PROGRAM PRG_RecipeManager
VAR
	fbLoadRecipe  	: FB_LoadRecipe;
    fbListFiles  	: FB_ListRecipeFiles;
	fbDeleteRecipe 	: FB_DeleteRecipe;
	fbSaveRecipe 	: FB_SaveRecipe;

    sPrefix      : STRING(64) := 'C:\TwinCAT\Recipes\';
    sFileName    : STRING(255);
	
	bDatagridRowsNaming		 : BOOL := FALSE;
	bClearAvailableFiles	 : BOOL := FALSE;
	bClearAvailableFilesDone : BOOL := FALSE;
	
	
		
	i	: INT;
	
	
END_VAR

VAR_INPUT
	bDatagridToRecipeDone	: BOOL := FALSE;
END_VAR

//Naming the datagrid 1st column with the names in the HMI Recipe Screen just once
IF NOT bDatagridRowsNaming THEN
	ACT_DatagridsRowNaming();
END_IF

// <Load button> ############# Look up for the recipe files in the folder and fill up the GVL_Recipe.aAvailableFiles[]. ######################### 
IF GVL_HMI.bRefreshRecipeList THEN
	//GVL_HMI.bRecipeCorrectLoaded := FALSE;
	//GVL_HMI.bRecipeLoadFailed := FALSE;
	bClearAvailableFiles := TRUE;
	IF bClearAvailableFilesDone THEN
		fbListFiles(bExecute := TRUE);
	END_IF
ELSE
	bClearAvailableFiles := FALSE;
	bClearAvailableFilesDone := FALSE;
    fbListFiles(bExecute := FALSE);
END_IF

// Clear the Available files datagrid in the load file popup
IF bClearAvailableFiles THEN
	ACT_ClearAvailableFiles();
END_IF

// Reset load actions once its done
IF fbListFiles.bDone THEN
	GVL_HMI.bRefreshRecipeList := FALSE;
END_IF

 //Reset file name
sFileName := '';

// Run the loading recipe from selected row in the recipe load popup
sFileName := CONCAT(sPrefix, CONCAT(GVL_Recipe.sSelectedRecipeName, '.json')); // File naming assemble for the selected row in the recipe load popup
fbLoadRecipe( sFileName := sFileName, bExecute := GVL_HMI.bRecipeLoadFromFile AND  DB_Query.timerVD.Q );


IF fbLoadRecipe.bError THEN
	GVL_HMI.bRecipeLoadFailed := TRUE;
	//GVL_HMI.bRecipeLoadFromFile := FALSE;
END_IF

// After the recipe loading, reseting and setting the flags
IF NOT fbLoadRecipe.bBusy AND NOT fbLoadRecipe.bError AND GVL_HMI.bRecipeLoadFromFile AND DB_Query.timerVD.Q THEN
	GVL_HMI.bRecipeCorrectLoaded := TRUE;
	GVL_HMI.bRecipeLoadFromFile := FALSE;
	DB_Query.timerVD(in:= FALSE);
	ACT_ClearStActiveRecipe(); //Clears the Active Recipe
END_IF
// <\Load button> ############# END ##############

// <Save Button> ############# Fill stCurrentRecipe from HMI datagrids if save button is pressed ########################
IF GVL_HMI.bRecipeSaveButton THEN
	ACT_DatagridToRecipe();
	IF bDatagridToRecipeDone THEN
		fbSaveRecipe(bExecute := TRUE, sUser := GVL_HMI.stRecipeInfo.sCreatedBy);
		IF fbSaveRecipe.bDone AND NOT fbSaveRecipe.bError THEN
			GVL_HMI.stRecipeInfo.iRevision := GVL_Recipe.stCurrentRecipe.stInfo.iRevision; //Update the datagrid revision that does not come from the grid
			fbSaveRecipe(bExecute := FALSE);
			GVL_HMI.bRecipeSaveDone := TRUE; //Response Success flag to HMI
			GVL_HMI.bRecipeSaveButton := FALSE;	
			bDatagridToRecipeDone := FALSE;
			ACT_ClearStActiveRecipe(); //Clears the Active Recipe
			ELSE IF fbSaveRecipe.bError THEN
				GVL_HMI.bRecipeSaveError := TRUE; //Response Error flag to HMI
			END_IF
		END_IF
		
	END_IF
END_IF
// <\Save Button> ############# END ########################

// <Cancel Button> ############# Reload the datagrids with the recipe in stCurrentRecipe if the bt cancel is pressed during new recipe ########################
IF GVL_HMI.bReloadRecipeDatagrids THEN
	ACT_RecipeToDatagrid();
END_IF
// <\Cancel Button> ############# END ########################

// <Activate Button> ############# Transfer data from stCurrentRecipe for stActivatedRecipe witch will be used on the cycle  ########################
IF GVL_HMI.bRecipeActivateButton THEN
	GVL_Recipe.stActiveRecipe := GVL_Recipe.stCurrentRecipe; //Only fill stActiveRecipe if button Activate was pressed on hmi. 
	IF GVL_Recipe.stCurrentRecipe.stInfo.sMethodName <> '' THEN
		GVL_HMI.bRecipeActivateDone := TRUE;
		GVL_Recipe.bIsThereRecipeActivated := TRUE;
	ELSE
		GVL_HMI.bRecipeActivateError := TRUE;
	END_IF
	
END_IF
// <\Activate Button> ############# END ########################

// <Delete Button> ############# Moves the loaded Recipe file from the root folder for the _deleted folder ########################
IF GVL_HMI.bDeleteRecipeButton THEN
	ACT_PopulateDeleteRecipeInfo();
	GVL_HMI.bDeleteRecipeDone := FALSE;
	GVL_HMI.bDeleteRecipeError := FALSE;
END_IF

fbDeleteRecipe(bExecute := GVL_HMI.bDeleteRecipeConfirm, stFileInfo := GVL_HMI.stDeleteRecipeInfo);

IF fbDeleteRecipe.bDone THEN
	IF NOT fbDeleteRecipe.bError THEN 
		ACT_ClearStCurrentRecipe();
		ACT_ClearHMIDatagrids();
		ACT_ClearStActiveRecipe(); //Clears the Active Recipe
		GVL_HMI.bDeleteRecipeConfirm := FALSE;
		GVL_HMI.bDeleteRecipeDone := TRUE;
	ELSE 
		GVL_HMI.bDeleteRecipeError := TRUE;
	END_IF
END_IF

// <\Delete Button> ############# END ########################

ACTION ACT_ClearAvailableFiles:
//Clear the GVL_Recipe.aAvailableFiles, witch is the list files datagrid data source
IF NOT bClearAvailableFilesDone THEN
	FOR i := 1 TO 50 DO
		GVL_HMI.aAvailableFiles[i].sFileName := '';
		GVL_HMI.aAvailableFiles[i].sMethodName := '';
		GVL_HMI.aAvailableFiles[i].sCreatedBy := '';
		GVL_HMI.aAvailableFiles[i].iRevision := 0;
		GVL_HMI.aAvailableFiles[i].dtLastModified := DT#1970-01-01-00:00;
		GVL_HMI.aAvailableFiles[i].dCreationDate := D#1970-01-01;
	END_FOR
	
	IF i >= 50 THEN
		bClearAvailableFilesDone := TRUE;
	END_IF
END_IF
END_ACTION

ACTION ACT_ClearHMIDatagrids:
//Clear the arrays that are binding with the datagrids source on recipe HMI content
//Recipe Info fields
GVL_HMI.stRecipeInfo.dCreationDate := D#1970-01-01;
GVL_HMI.stRecipeInfo.iRevision := 0;
GVL_HMI.stRecipeInfo.sCreatedBy := '';
GVL_HMI.stRecipeInfo.sMethodName := '';

//Solvents and Times datagrid
FOR i := 1 TO 3 DO
	GVL_HMI.aSolventAndTimesRows[i].Rinse1 := 0;
	GVL_HMI.aSolventAndTimesRows[i].Rinse2 := 0;
	GVL_HMI.aSolventAndTimesRows[i].Wash1 := 0;
	GVL_HMI.aSolventAndTimesRows[i].Wash2 := 0;
END_FOR

//Volumes datagrid
FOR i := 1 TO 10 DO
	GVL_HMI.aVolumeRows[i].Rinse1 := 0;
	GVL_HMI.aVolumeRows[i].Rinse2 := 0;
	GVL_HMI.aVolumeRows[i].Wash1 := 0;
	GVL_HMI.aVolumeRows[i].Wash2 := 0;
END_FOR

//Other Parameters datagrid
FOR i := 1 TO 8 DO
	GVL_HMI.aOtherParamsRows[i].Value := 0;
END_FOR
END_ACTION

ACTION ACT_ClearStActiveRecipe:
//Clear Flags 
GVL_Recipe.bIsThereRecipeActivated := FALSE;
GVL_HMI.bRecipeActivateDone := FALSE;
GVL_HMI.bRecipeActivateError := FALSE;
//Clears the array stCurrentRecipe 
//Info
GVL_Recipe.stActiveRecipe.stInfo.dCreationDate := D#1970-01-01;
GVL_Recipe.stActiveRecipe.stInfo.iRevision := 0;
GVL_Recipe.stActiveRecipe.stInfo.sCreatedBy := '';
GVL_Recipe.stActiveRecipe.stInfo.sMethodName := '';


//Other Parameters
GVL_Recipe.stActiveRecipe.stOtherParams.iVialsToFill := 0;
GVL_Recipe.stActiveRecipe.stOtherParams.rVial1FillVol := 0;
GVL_Recipe.stActiveRecipe.stOtherParams.rVialPrimeVol := 0;
GVL_Recipe.stActiveRecipe.stOtherParams.rVials2_4FillVol := 0;
GVL_Recipe.stActiveRecipe.stOtherParams.tAgitate1Time := T#0S;
GVL_Recipe.stActiveRecipe.stOtherParams.tAgitate2Time := T#0S;
GVL_Recipe.stActiveRecipe.stOtherParams.tAirDryTime := T#0S;
GVL_Recipe.stActiveRecipe.stOtherParams.tSoakTime := T#0S;

FOR i := 1 TO 4 DO
	//Solvents and Times
	GVL_Recipe.stActiveRecipe.stSolventsTimes.aSolventN[i] := 0;
	GVL_Recipe.stActiveRecipe.stSolventsTimes.aTime[i] := T#0S;
	GVL_Recipe.stActiveRecipe.stSolventsTimes.aVelocity[i] := 0;
	
	//Volumes
	GVL_Recipe.stActiveRecipe.stVolumes.aF_Volume[i] := 0;
	GVL_Recipe.stActiveRecipe.stVolumes.aS0_Volume[i] := 0;
	GVL_Recipe.stActiveRecipe.stVolumes.aS1_Volume[i] := 0;
	GVL_Recipe.stActiveRecipe.stVolumes.aS2_Volume[i] := 0;
	GVL_Recipe.stActiveRecipe.stVolumes.aS3_Volume[i] := 0;
	GVL_Recipe.stActiveRecipe.stVolumes.aS4_Volume[i] := 0;
	GVL_Recipe.stActiveRecipe.stVolumes.aS5_Volume[i] := 0;
	GVL_Recipe.stActiveRecipe.stVolumes.aS6_Volume[i] := 0;
	GVL_Recipe.stActiveRecipe.stVolumes.aS7_Volume[i] := 0;
	GVL_Recipe.stActiveRecipe.stVolumes.aT_IC_Volume[i] := 0;
END_FOR
END_ACTION

ACTION ACT_ClearStCurrentRecipe:
//Clears the array stCurrentRecipe 
//Info
GVL_Recipe.stCurrentRecipe.stInfo.dCreationDate := D#1970-01-01;
GVL_Recipe.stCurrentRecipe.stInfo.iRevision := 0;
GVL_Recipe.stCurrentRecipe.stInfo.sCreatedBy := '';
GVL_Recipe.stCurrentRecipe.stInfo.sMethodName := '';

//Other Parameters
GVL_Recipe.stCurrentRecipe.stOtherParams.iVialsToFill := 0;
GVL_Recipe.stCurrentRecipe.stOtherParams.rVial1FillVol := 0;
GVL_Recipe.stCurrentRecipe.stOtherParams.rVialPrimeVol := 0;
GVL_Recipe.stCurrentRecipe.stOtherParams.rVials2_4FillVol := 0;
GVL_Recipe.stCurrentRecipe.stOtherParams.tAgitate1Time := T#0S;
GVL_Recipe.stCurrentRecipe.stOtherParams.tAgitate2Time := T#0S;
GVL_Recipe.stCurrentRecipe.stOtherParams.tAirDryTime := T#0S;
GVL_Recipe.stCurrentRecipe.stOtherParams.tSoakTime := T#0S;

FOR i := 1 TO 4 DO
	//Solvents and Times
	GVL_Recipe.stCurrentRecipe.stSolventsTimes.aSolventN[i] := 0;
	GVL_Recipe.stCurrentRecipe.stSolventsTimes.aTime[i] := T#0S;
	GVL_Recipe.stCurrentRecipe.stSolventsTimes.aVelocity[i] := 0;
	
	//Volumes
	GVL_Recipe.stCurrentRecipe.stVolumes.aF_Volume[i] := 0;
	GVL_Recipe.stCurrentRecipe.stVolumes.aS0_Volume[i] := 0;
	GVL_Recipe.stCurrentRecipe.stVolumes.aS1_Volume[i] := 0;
	GVL_Recipe.stCurrentRecipe.stVolumes.aS2_Volume[i] := 0;
	GVL_Recipe.stCurrentRecipe.stVolumes.aS3_Volume[i] := 0;
	GVL_Recipe.stCurrentRecipe.stVolumes.aS4_Volume[i] := 0;
	GVL_Recipe.stCurrentRecipe.stVolumes.aS5_Volume[i] := 0;
	GVL_Recipe.stCurrentRecipe.stVolumes.aS6_Volume[i] := 0;
	GVL_Recipe.stCurrentRecipe.stVolumes.aS7_Volume[i] := 0;
	GVL_Recipe.stCurrentRecipe.stVolumes.aT_IC_Volume[i] := 0;
END_FOR
END_ACTION

ACTION ACT_DatagridsRowNaming:
//Naming the HMI Recipe Screen Datagrid rows
//TcHmiDatagrid_SolventAndTimes
GVL_HMI.aSolventAndTimesRows[1].Parameter := 'Solvent #';
GVL_HMI.aSolventAndTimesRows[2].Parameter := 'Time';
GVL_HMI.aSolventAndTimesRows[3].Parameter := 'Velocity';

//TcHmiDatagrid_Volumes
GVL_HMI.aVolumeRows[1].Stage := 'T/IC';
GVL_HMI.aVolumeRows[2].Stage := 'S0';
GVL_HMI.aVolumeRows[3].Stage := 'S1';
GVL_HMI.aVolumeRows[4].Stage := 'S2';
GVL_HMI.aVolumeRows[5].Stage := 'S3';
GVL_HMI.aVolumeRows[6].Stage := 'S4';
GVL_HMI.aVolumeRows[7].Stage := 'S5';
GVL_HMI.aVolumeRows[8].Stage := 'S6';
GVL_HMI.aVolumeRows[9].Stage := 'S7';
GVL_HMI.aVolumeRows[10].Stage := 'F';

//TcHmiDatagrid_OtherParams
GVL_HMI.aOtherParamsRows[1].Parameter := 'Soak Time';
GVL_HMI.aOtherParamsRows[2].Parameter := 'Agitate 1 Time';
GVL_HMI.aOtherParamsRows[3].Parameter := 'Agitate 2 Time';
GVL_HMI.aOtherParamsRows[4].Parameter := 'Vials to Fill';
GVL_HMI.aOtherParamsRows[5].Parameter := 'Vial Prime Vol';
GVL_HMI.aOtherParamsRows[6].Parameter := 'Vial 1 Fill Vol';
GVL_HMI.aOtherParamsRows[7].Parameter := 'Vials 2-4 Fill Vol';
GVL_HMI.aOtherParamsRows[8].Parameter := 'Air Dry Time';
//TcHmiDatagrid_OtherParams - Data Units
GVL_HMI.aOtherParamsRows[1].Units     := 'sec';
GVL_HMI.aOtherParamsRows[2].Units     := 'sec';
GVL_HMI.aOtherParamsRows[3].Units     := 'sec';
GVL_HMI.aOtherParamsRows[4].Units     := 'unit';
GVL_HMI.aOtherParamsRows[5].Units     := 'ml';
GVL_HMI.aOtherParamsRows[6].Units     := 'ml';
GVL_HMI.aOtherParamsRows[7].Units     := 'ml';
GVL_HMI.aOtherParamsRows[8].Units     := 'sec';

//Finish the naming
bDatagridRowsNaming := TRUE;
END_ACTION

ACTION ACT_DatagridToRecipe:
IF NOT bDatagridToRecipeDone THEN
	// ---- Commit RecipeInfo ----	
	GVL_Recipe.stCurrentRecipe.stInfo.sCreatedBy := GVL_HMI.stRecipeInfo.sCreatedBy;
	GVL_Recipe.stCurrentRecipe.stInfo.sMethodName := GVL_HMI.stRecipeInfo.sMethodName;
	

	// ---- Commit SolventAndTimes ----
	FOR i := 1 TO 4 DO // 1: Rinse1, 2: Rinse2, 3: Wash1, 4: Wash2
		// Solvent #
		CASE i OF
			1: GVL_Recipe.stCurrentRecipe.stSolventsTimes.aSolventN[i] := TO_USINT(GVL_HMI.aSolventAndTimesRows[1].Rinse1);
			2: GVL_Recipe.stCurrentRecipe.stSolventsTimes.aSolventN[i] := TO_USINT(GVL_HMI.aSolventAndTimesRows[1].Rinse2);
			3: GVL_Recipe.stCurrentRecipe.stSolventsTimes.aSolventN[i] := TO_USINT(GVL_HMI.aSolventAndTimesRows[1].Wash1);
			4: GVL_Recipe.stCurrentRecipe.stSolventsTimes.aSolventN[i] := TO_USINT(GVL_HMI.aSolventAndTimesRows[1].Wash2);
		END_CASE;
		// Time (convertendo para TIME)
		CASE i OF
			1: GVL_Recipe.stCurrentRecipe.stSolventsTimes.aTime[i] := DWORD_TO_TIME(GVL_HMI.aSolventAndTimesRows[2].Rinse1 * 1000);
			2: GVL_Recipe.stCurrentRecipe.stSolventsTimes.aTime[i] := DWORD_TO_TIME(GVL_HMI.aSolventAndTimesRows[2].Rinse2 * 1000);
			3: GVL_Recipe.stCurrentRecipe.stSolventsTimes.aTime[i] := DWORD_TO_TIME(GVL_HMI.aSolventAndTimesRows[2].Wash1 * 1000);
			4: GVL_Recipe.stCurrentRecipe.stSolventsTimes.aTime[i] := DWORD_TO_TIME(GVL_HMI.aSolventAndTimesRows[2].Wash2 * 1000);
		END_CASE;
		// Velocity
		CASE i OF
			1: GVL_Recipe.stCurrentRecipe.stSolventsTimes.aVelocity[i] := GVL_HMI.aSolventAndTimesRows[3].Rinse1;
			2: GVL_Recipe.stCurrentRecipe.stSolventsTimes.aVelocity[i] := GVL_HMI.aSolventAndTimesRows[3].Rinse2;
			3: GVL_Recipe.stCurrentRecipe.stSolventsTimes.aVelocity[i] := GVL_HMI.aSolventAndTimesRows[3].Wash1;
			4: GVL_Recipe.stCurrentRecipe.stSolventsTimes.aVelocity[i] := GVL_HMI.aSolventAndTimesRows[3].Wash2;
		END_CASE;
	END_FOR
	
	// ---- Commit Volumes ----
	// Cada linha do aVolumesRows corresponde a um array do struct
	// Ordem: 1:T_IC, 2:S0, 3:S1, 4:S2, 5:S3, 6:S4, 7:S5, 8:S6, 9:S7, 10:F
	FOR i := 1 TO 4 DO // Rinse1, Rinse2, Wash1, Wash2
		// T_IC
		CASE i OF
			1: GVL_Recipe.stCurrentRecipe.stVolumes.aT_IC_Volume[i] := GVL_HMI.aVolumeRows[1].Rinse1;
			2: GVL_Recipe.stCurrentRecipe.stVolumes.aT_IC_Volume[i] := GVL_HMI.aVolumeRows[1].Rinse2;
			3: GVL_Recipe.stCurrentRecipe.stVolumes.aT_IC_Volume[i] := GVL_HMI.aVolumeRows[1].Wash1;
			4: GVL_Recipe.stCurrentRecipe.stVolumes.aT_IC_Volume[i] := GVL_HMI.aVolumeRows[1].Wash2;
		END_CASE;
		// S0
		CASE i OF
			1: GVL_Recipe.stCurrentRecipe.stVolumes.aS0_Volume[i] := GVL_HMI.aVolumeRows[2].Rinse1;
			2: GVL_Recipe.stCurrentRecipe.stVolumes.aS0_Volume[i] := GVL_HMI.aVolumeRows[2].Rinse2;
			3: GVL_Recipe.stCurrentRecipe.stVolumes.aS0_Volume[i] := GVL_HMI.aVolumeRows[2].Wash1;
			4: GVL_Recipe.stCurrentRecipe.stVolumes.aS0_Volume[i] := GVL_HMI.aVolumeRows[2].Wash2;
		END_CASE;
		// S1 
		CASE i OF
			1: GVL_Recipe.stCurrentRecipe.stVolumes.aS1_Volume[i] := GVL_HMI.aVolumeRows[3].Rinse1;
			2: GVL_Recipe.stCurrentRecipe.stVolumes.aS1_Volume[i] := GVL_HMI.aVolumeRows[3].Rinse2;
			3: GVL_Recipe.stCurrentRecipe.stVolumes.aS1_Volume[i] := GVL_HMI.aVolumeRows[3].Wash1;
			4: GVL_Recipe.stCurrentRecipe.stVolumes.aS1_Volume[i] := GVL_HMI.aVolumeRows[3].Wash2;
		END_CASE;
		// S2
		CASE i OF
			1: GVL_Recipe.stCurrentRecipe.stVolumes.aS2_Volume[i] := GVL_HMI.aVolumeRows[4].Rinse1;
			2: GVL_Recipe.stCurrentRecipe.stVolumes.aS2_Volume[i] := GVL_HMI.aVolumeRows[4].Rinse2;
			3: GVL_Recipe.stCurrentRecipe.stVolumes.aS2_Volume[i] := GVL_HMI.aVolumeRows[4].Wash1;
			4: GVL_Recipe.stCurrentRecipe.stVolumes.aS2_Volume[i] := GVL_HMI.aVolumeRows[4].Wash2;
		END_CASE;
		CASE i OF
			1: GVL_Recipe.stCurrentRecipe.stVolumes.aS3_Volume[i] := GVL_HMI.aVolumeRows[5].Rinse1;
			2: GVL_Recipe.stCurrentRecipe.stVolumes.aS3_Volume[i] := GVL_HMI.aVolumeRows[5].Rinse2;
			3: GVL_Recipe.stCurrentRecipe.stVolumes.aS3_Volume[i] := GVL_HMI.aVolumeRows[5].Wash1;
			4: GVL_Recipe.stCurrentRecipe.stVolumes.aS3_Volume[i] := GVL_HMI.aVolumeRows[5].Wash2;
		END_CASE;
		CASE i OF
			1: GVL_Recipe.stCurrentRecipe.stVolumes.aS4_Volume[i] := GVL_HMI.aVolumeRows[6].Rinse1;
			2: GVL_Recipe.stCurrentRecipe.stVolumes.aS4_Volume[i] := GVL_HMI.aVolumeRows[6].Rinse2;
			3: GVL_Recipe.stCurrentRecipe.stVolumes.aS4_Volume[i] := GVL_HMI.aVolumeRows[6].Wash1;
			4: GVL_Recipe.stCurrentRecipe.stVolumes.aS4_Volume[i] := GVL_HMI.aVolumeRows[6].Wash2;
		END_CASE;
		CASE i OF
			1: GVL_Recipe.stCurrentRecipe.stVolumes.aS5_Volume[i] := GVL_HMI.aVolumeRows[7].Rinse1;
			2: GVL_Recipe.stCurrentRecipe.stVolumes.aS5_Volume[i] := GVL_HMI.aVolumeRows[7].Rinse2;
			3: GVL_Recipe.stCurrentRecipe.stVolumes.aS5_Volume[i] := GVL_HMI.aVolumeRows[7].Wash1;
			4: GVL_Recipe.stCurrentRecipe.stVolumes.aS5_Volume[i] := GVL_HMI.aVolumeRows[7].Wash2;
		END_CASE;
		CASE i OF
			1: GVL_Recipe.stCurrentRecipe.stVolumes.aS6_Volume[i] := GVL_HMI.aVolumeRows[8].Rinse1;
			2: GVL_Recipe.stCurrentRecipe.stVolumes.aS6_Volume[i] := GVL_HMI.aVolumeRows[8].Rinse2;
			3: GVL_Recipe.stCurrentRecipe.stVolumes.aS6_Volume[i] := GVL_HMI.aVolumeRows[8].Wash1;
			4: GVL_Recipe.stCurrentRecipe.stVolumes.aS6_Volume[i] := GVL_HMI.aVolumeRows[8].Wash2;
		END_CASE;
		CASE i OF
			1: GVL_Recipe.stCurrentRecipe.stVolumes.aS7_Volume[i] := GVL_HMI.aVolumeRows[9].Rinse1;
			2: GVL_Recipe.stCurrentRecipe.stVolumes.aS7_Volume[i] := GVL_HMI.aVolumeRows[9].Rinse2;
			3: GVL_Recipe.stCurrentRecipe.stVolumes.aS7_Volume[i] := GVL_HMI.aVolumeRows[9].Wash1;
			4: GVL_Recipe.stCurrentRecipe.stVolumes.aS7_Volume[i] := GVL_HMI.aVolumeRows[9].Wash2;
		END_CASE;
		CASE i OF
			1: GVL_Recipe.stCurrentRecipe.stVolumes.aF_Volume[i] := GVL_HMI.aVolumeRows[10].Rinse1;
			2: GVL_Recipe.stCurrentRecipe.stVolumes.aF_Volume[i] := GVL_HMI.aVolumeRows[10].Rinse2;
			3: GVL_Recipe.stCurrentRecipe.stVolumes.aF_Volume[i] := GVL_HMI.aVolumeRows[10].Wash1;
			4: GVL_Recipe.stCurrentRecipe.stVolumes.aF_Volume[i] := GVL_HMI.aVolumeRows[10].Wash2;
		END_CASE;
	END_FOR
	
	// ---- Commit OtherParams ----
	// Supondo a ordem das linhas conforme DataGrid (ajuste se necessário)
	GVL_Recipe.stCurrentRecipe.stOtherParams.tSoakTime        := TO_TIME(GVL_HMI.aOtherParamsRows[1].Value * 1000);
	GVL_Recipe.stCurrentRecipe.stOtherParams.tAgitate1Time    := TO_TIME(GVL_HMI.aOtherParamsRows[2].Value * 1000);
	GVL_Recipe.stCurrentRecipe.stOtherParams.tAgitate2Time    := TO_TIME(GVL_HMI.aOtherParamsRows[3].Value * 1000);
	GVL_Recipe.stCurrentRecipe.stOtherParams.iVialsToFill     := TO_USINT(GVL_HMI.aOtherParamsRows[4].Value);
	GVL_Recipe.stCurrentRecipe.stOtherParams.rVialPrimeVol    := GVL_HMI.aOtherParamsRows[5].Value;
	GVL_Recipe.stCurrentRecipe.stOtherParams.rVial1FillVol    := GVL_HMI.aOtherParamsRows[6].Value;
	GVL_Recipe.stCurrentRecipe.stOtherParams.rVials2_4FillVol := GVL_HMI.aOtherParamsRows[7].Value;
	GVL_Recipe.stCurrentRecipe.stOtherParams.tAirDryTime   	  := TO_TIME(GVL_HMI.aOtherParamsRows[8].Value * 1000);
	
	//reset flags
	
	i:=0;
	
	DB_Edit_Method(start:=TRUE);
	
	
END_IF
END_ACTION

ACTION ACT_PopulateDeleteRecipeInfo:
// Fill up the info fields for popup delete confirmation
GVL_HMI.stDeleteRecipeInfo.sCreatedBy := GVL_Recipe.stCurrentRecipe.stInfo.sCreatedBy;
GVL_HMI.stDeleteRecipeInfo.dCreationDate := GVL_Recipe.stCurrentRecipe.stInfo.dCreationDate;
GVL_HMI.stDeleteRecipeInfo.iRevision := GVL_Recipe.stCurrentRecipe.stInfo.iRevision;
GVL_HMI.stDeleteRecipeInfo.sMethodName := GVL_Recipe.stCurrentRecipe.stInfo.sMethodName;
GVL_HMI.stDeleteRecipeInfo.sFileName := GVL_Recipe.sSelectedRecipeName;

// Resets the flag
GVL_HMI.bDeleteRecipeButton := FALSE;
END_ACTION

ACTION ACT_RecipeToDatagrid:

// SolventAndTimes
GVL_HMI.aSolventAndTimesRows[1].Rinse1 := GVL_Recipe.stCurrentRecipe.stSolventsTimes.aSolventN[1];
GVL_HMI.aSolventAndTimesRows[1].Rinse2 := GVL_Recipe.stCurrentRecipe.stSolventsTimes.aSolventN[2];
GVL_HMI.aSolventAndTimesRows[1].Wash1  := GVL_Recipe.stCurrentRecipe.stSolventsTimes.aSolventN[3];
GVL_HMI.aSolventAndTimesRows[1].Wash2  := GVL_Recipe.stCurrentRecipe.stSolventsTimes.aSolventN[4];

GVL_HMI.aSolventAndTimesRows[2].Rinse1 := TO_INT(TIME_TO_DWORD(GVL_Recipe.stCurrentRecipe.stSolventsTimes.aTime[1])/1000);
GVL_HMI.aSolventAndTimesRows[2].Rinse2 := TO_INT(TIME_TO_DWORD(GVL_Recipe.stCurrentRecipe.stSolventsTimes.aTime[2])/1000);
GVL_HMI.aSolventAndTimesRows[2].Wash1  := TO_INT(TIME_TO_DWORD(GVL_Recipe.stCurrentRecipe.stSolventsTimes.aTime[3])/1000);
GVL_HMI.aSolventAndTimesRows[2].Wash2  := TO_INT(TIME_TO_DWORD(GVL_Recipe.stCurrentRecipe.stSolventsTimes.aTime[4])/1000);

GVL_HMI.aSolventAndTimesRows[3].Rinse1 := GVL_Recipe.stCurrentRecipe.stSolventsTimes.aVelocity[1];
GVL_HMI.aSolventAndTimesRows[3].Rinse2 := GVL_Recipe.stCurrentRecipe.stSolventsTimes.aVelocity[2];
GVL_HMI.aSolventAndTimesRows[3].Wash1  := GVL_Recipe.stCurrentRecipe.stSolventsTimes.aVelocity[3];
GVL_HMI.aSolventAndTimesRows[3].Wash2  := GVL_Recipe.stCurrentRecipe.stSolventsTimes.aVelocity[4];

// Volumes
GVL_HMI.aVolumeRows[1].Rinse1 := GVL_Recipe.stCurrentRecipe.stVolumes.aT_IC_Volume[1];
GVL_HMI.aVolumeRows[1].Rinse2 := GVL_Recipe.stCurrentRecipe.stVolumes.aT_IC_Volume[2];
GVL_HMI.aVolumeRows[1].Wash1  := GVL_Recipe.stCurrentRecipe.stVolumes.aT_IC_Volume[3];
GVL_HMI.aVolumeRows[1].Wash2  := GVL_Recipe.stCurrentRecipe.stVolumes.aT_IC_Volume[4];

GVL_HMI.aVolumeRows[2].Rinse1 := GVL_Recipe.stCurrentRecipe.stVolumes.aS0_Volume[1];
GVL_HMI.aVolumeRows[2].Rinse2 := GVL_Recipe.stCurrentRecipe.stVolumes.aS0_Volume[2];
GVL_HMI.aVolumeRows[2].Wash1  := GVL_Recipe.stCurrentRecipe.stVolumes.aS0_Volume[3];
GVL_HMI.aVolumeRows[2].Wash2  := GVL_Recipe.stCurrentRecipe.stVolumes.aS0_Volume[4];

GVL_HMI.aVolumeRows[3].Rinse1 := GVL_Recipe.stCurrentRecipe.stVolumes.aS1_Volume[1];
GVL_HMI.aVolumeRows[3].Rinse2 := GVL_Recipe.stCurrentRecipe.stVolumes.aS1_Volume[2];
GVL_HMI.aVolumeRows[3].Wash1  := GVL_Recipe.stCurrentRecipe.stVolumes.aS1_Volume[3];
GVL_HMI.aVolumeRows[3].Wash2  := GVL_Recipe.stCurrentRecipe.stVolumes.aS1_Volume[4];

GVL_HMI.aVolumeRows[4].Rinse1 := GVL_Recipe.stCurrentRecipe.stVolumes.aS2_Volume[1];
GVL_HMI.aVolumeRows[4].Rinse2 := GVL_Recipe.stCurrentRecipe.stVolumes.aS2_Volume[2];
GVL_HMI.aVolumeRows[4].Wash1  := GVL_Recipe.stCurrentRecipe.stVolumes.aS2_Volume[3];
GVL_HMI.aVolumeRows[4].Wash2  := GVL_Recipe.stCurrentRecipe.stVolumes.aS2_Volume[4];

GVL_HMI.aVolumeRows[5].Rinse1 := GVL_Recipe.stCurrentRecipe.stVolumes.aS3_Volume[1];
GVL_HMI.aVolumeRows[5].Rinse2 := GVL_Recipe.stCurrentRecipe.stVolumes.aS3_Volume[2];
GVL_HMI.aVolumeRows[5].Wash1  := GVL_Recipe.stCurrentRecipe.stVolumes.aS3_Volume[3];
GVL_HMI.aVolumeRows[5].Wash2  := GVL_Recipe.stCurrentRecipe.stVolumes.aS3_Volume[4];

GVL_HMI.aVolumeRows[6].Rinse1 := GVL_Recipe.stCurrentRecipe.stVolumes.aS4_Volume[1];
GVL_HMI.aVolumeRows[6].Rinse2 := GVL_Recipe.stCurrentRecipe.stVolumes.aS4_Volume[2];
GVL_HMI.aVolumeRows[6].Wash1  := GVL_Recipe.stCurrentRecipe.stVolumes.aS4_Volume[3];
GVL_HMI.aVolumeRows[6].Wash2  := GVL_Recipe.stCurrentRecipe.stVolumes.aS4_Volume[4];

GVL_HMI.aVolumeRows[7].Rinse1 := GVL_Recipe.stCurrentRecipe.stVolumes.aS5_Volume[1];
GVL_HMI.aVolumeRows[7].Rinse2 := GVL_Recipe.stCurrentRecipe.stVolumes.aS5_Volume[2];
GVL_HMI.aVolumeRows[7].Wash1  := GVL_Recipe.stCurrentRecipe.stVolumes.aS5_Volume[3];
GVL_HMI.aVolumeRows[7].Wash2  := GVL_Recipe.stCurrentRecipe.stVolumes.aS5_Volume[4];

GVL_HMI.aVolumeRows[8].Rinse1 := GVL_Recipe.stCurrentRecipe.stVolumes.aS6_Volume[1];
GVL_HMI.aVolumeRows[8].Rinse2 := GVL_Recipe.stCurrentRecipe.stVolumes.aS6_Volume[2];
GVL_HMI.aVolumeRows[8].Wash1  := GVL_Recipe.stCurrentRecipe.stVolumes.aS6_Volume[3];
GVL_HMI.aVolumeRows[8].Wash2  := GVL_Recipe.stCurrentRecipe.stVolumes.aS6_Volume[4];

GVL_HMI.aVolumeRows[9].Rinse1 := GVL_Recipe.stCurrentRecipe.stVolumes.aS7_Volume[1];
GVL_HMI.aVolumeRows[9].Rinse2 := GVL_Recipe.stCurrentRecipe.stVolumes.aS7_Volume[2];
GVL_HMI.aVolumeRows[9].Wash1  := GVL_Recipe.stCurrentRecipe.stVolumes.aS7_Volume[3];
GVL_HMI.aVolumeRows[9].Wash2  := GVL_Recipe.stCurrentRecipe.stVolumes.aS7_Volume[4];

GVL_HMI.aVolumeRows[10].Rinse1 := GVL_Recipe.stCurrentRecipe.stVolumes.aF_Volume[1];
GVL_HMI.aVolumeRows[10].Rinse2 := GVL_Recipe.stCurrentRecipe.stVolumes.aF_Volume[2];
GVL_HMI.aVolumeRows[10].Wash1  := GVL_Recipe.stCurrentRecipe.stVolumes.aF_Volume[3];
GVL_HMI.aVolumeRows[10].Wash2  := GVL_Recipe.stCurrentRecipe.stVolumes.aF_Volume[4];

// --- Outros Params ---
GVL_HMI.aOtherParamsRows[1].Value := UDINT_TO_REAL(TIME_TO_DWORD(GVL_Recipe.stCurrentRecipe.stOtherParams.tSoakTime)/1000);
GVL_HMI.aOtherParamsRows[2].Value := UDINT_TO_REAL(TIME_TO_DWORD(GVL_Recipe.stCurrentRecipe.stOtherParams.tAgitate1Time)/1000);
GVL_HMI.aOtherParamsRows[3].Value := UDINT_TO_REAL(TIME_TO_DWORD(GVL_Recipe.stCurrentRecipe.stOtherParams.tAgitate2Time)/1000);
GVL_HMI.aOtherParamsRows[4].Value := GVL_Recipe.stCurrentRecipe.stOtherParams.iVialsToFill;
GVL_HMI.aOtherParamsRows[5].Value := GVL_Recipe.stCurrentRecipe.stOtherParams.rVialPrimeVol;
GVL_HMI.aOtherParamsRows[6].Value := GVL_Recipe.stCurrentRecipe.stOtherParams.rVial1FillVol;
GVL_HMI.aOtherParamsRows[7].Value := GVL_Recipe.stCurrentRecipe.stOtherParams.rVials2_4FillVol;
GVL_HMI.aOtherParamsRows[8].Value := UDINT_TO_REAL(TIME_TO_DWORD(GVL_Recipe.stCurrentRecipe.stOtherParams.tAirDryTime)/1000);

//Flag to initiate the save fb
GVL_HMI.bReloadRecipeDatagrids  := FALSE;
END_ACTION

END_PROGRAM

(* stored: Version 1.1.0.1, ProductVersion 3.1.4024.15
   POU PRG_RecipeManager: Id {f4641f87-7b16-4bb3-8169-d73676afbb75}, SpecialFunc None
   Action ACT_ClearAvailableFiles: Id {69c4ef56-ea89-4269-bd3f-37b671659ed2}
   Action ACT_ClearHMIDatagrids: Id {ac68110a-010b-4d2e-a48f-41c3d72a6a58}
   Action ACT_ClearStActiveRecipe: Id {7d7b713d-eb13-4628-ac48-368a599d0c01}
   Action ACT_ClearStCurrentRecipe: Id {015909d4-6612-4235-8058-47c7ae45226c}
   Action ACT_DatagridsRowNaming: Id {7a5f0b3d-52d7-4ce2-b6cd-e160802e7ce0}
   Action ACT_DatagridToRecipe: Id {d800e175-fa01-48f3-8ed7-dde5a40976cb}
   Action ACT_PopulateDeleteRecipeInfo: Id {441531cc-5411-489e-b8c8-b1846bd52885}
   Action ACT_RecipeToDatagrid: Id {947174eb-de1f-4e9d-b1cf-e0d4928d41c5} *)
